TYPE ST_GCSingleProcessCycleRecord :
STRUCT
	Result : E_GCSingleProcessResult;
	FailedStage : E_GCSingleProcessStage;
	FailedAxis : E_GCSingleProcessAxis;
	TotalActualTime : TIME;
	StageTiming : ST_GCSingleProcessStageTimings;
END_STRUCT
END_TYPE

(* stored: Version 1.1.0.1, ProductVersion 3.1.4026.18
   DUT ST_GCSingleProcessCycleRecord: Id {3a36c780-9736-474d-b450-1ac197e48da4} *)
